KUKA KRL program: kuka_eki_command_serverB.sub, kuka_eki_command_serverB.dat

--- kuka_eki_command_serverB.sub ---
&ACCESS RVO1
&PARAM EDITMASK = *
&PARAM TEMPLATE = C:\KRC\Roboter\Template\submit
def kuka_eki_command_serverB()
   ;FOLD DECLARATIONS
   ;FOLD USER DECL
   ; local vairable declarations
   decl int elements_read

   eki_hw_iface_init() ; socket connection

   parameters[1] = $POS_ACT.X
   parameters[2] = $POS_ACT.Y
   parameters[3] = $POS_ACT.Z
   parameters[4] = $POS_ACT.A
   parameters[5] = $POS_ACT.B
   parameters[6] = $POS_ACT.C

   loop
      instruction_code = 0 ; reset instruction code to default
      elements_read = eki_hw_iface_get()  ; Get new command from buffer

      SWITCH (instruction_code)
      CASE 1
         ; cartesian motion XYZ command, phrase parameters into global variable cartesian_target
         cartesian_target.X = parameters[1]
         cartesian_target.Y = parameters[2]
         cartesian_target.Z = parameters[3]
         MsgNotify("Cartesian target XYZ command received and set",,,,)

      CASE 2
         ; cartesian motion XYZABC command
         cartesian_target.X = parameters[1]
         cartesian_target.Y = parameters[2]
         cartesian_target.Z = parameters[3]
         cartesian_target.A = parameters[4]
         cartesian_target.B = parameters[5]
         cartesian_target.C = parameters[6]

      CASE 3
         ; whether motion complete (0/1)
         json_motion_complete = parameters[1]

      CASE 4
         ; set linear velocity
         $VEL.CP = parameters[1]

      CASE 5
         ; set swivel velocity
         $VEL.ORI1 = parameters[1]

      CASE 6
         ; set swivel velocity
         $VEL.ORI2 = parameters[1]

      CASE 7
         LaserOff()
      CASE 8
         LaserOn()
      CASE 9
         LaserEnd()
      CASE 10
         LaserStart()
      CASE 11
         $ANOUT[1] = parameters[1] ; set laser power
      CASE 12
         $TOOL=TOOL_DATA[parameters[1]] ; set tool
      CASE 13
         $BASE.X = parameters[1]
         $BASE.Y = parameters[2]
         $BASE.Z = parameters[3]
         $BASE.A = parameters[4]
         $BASE.B = parameters[5]
         $BASE.C = parameters[6]
      CASE 14
         ;wait time between move
         wait_time = parameters[1]


      DEFAULT
         cartesian_target.X = $POS_ACT.X
         cartesian_target.Y = $POS_ACT.Y
         cartesian_target.Z = $POS_ACT.Z
         cartesian_target.A = $POS_ACT.A
         cartesian_target.B = $POS_ACT.B
         cartesian_target.C = $POS_ACT.C
      ENDSWITCH
   endloop


end



def eki_hw_iface_init()
   decl eki_status eki_ret

   ; Setup interrupts
   ; Interrupt 15 - Connection cleanup on client disconnect
   global interrupt decl 15 when $flag[1]==false do eki_hw_iface_reset()
   interrupt on 15
   ; Interrupt 16 - Timer interrupt for periodic state transmission
   global interrupt decl 16 when $timer_flag[1]==true do eki_hw_iface_send()
   interrupt on 16
   wait sec 0.012          ; Wait for next interpolation cycle
   $timer[1] = -200        ; Time in [ms] before first interrupt call
   $timer_stop[1] = false  ; Start timer 1

   ; Create and open EKI interface
   eki_ret = eki_init("EkiCommandServerB")
   eki_ret = eki_open("EkiCommandServerB")
   MsgNotify("ROS connection established",,,,)
end



def eki_hw_iface_send()
   decl eki_status eki_ret

   if $flag[1] then  ; If connection alive
      ; Load state values into xml structure
      ; position
      eki_ret = eki_setreal("EkiCommandServerB", "RobotState/Pos/@A1", $axis_act_meas.a1)
      eki_ret = eki_setreal("EkiCommandServerB", "RobotState/Pos/@A2", $axis_act_meas.a2)
      eki_ret = eki_setreal("EkiCommandServerB", "RobotState/Pos/@A3", $axis_act_meas.a3)
      eki_ret = eki_setreal("EkiCommandServerB", "RobotState/Pos/@A4", $axis_act_meas.a4)
      eki_ret = eki_setreal("EkiCommandServerB", "RobotState/Pos/@A5", $axis_act_meas.a5)
      eki_ret = eki_setreal("EkiCommandServerB", "RobotState/Pos/@A6", $axis_act_meas.a6)

      eki_ret = eki_setreal("EkiCommandServerB", "RobotState/Eff/@A1", $torque_axis_act[1])
      eki_ret = eki_setreal("EkiCommandServerB", "RobotState/Eff/@A2", $torque_axis_act[2])
      eki_ret = eki_setreal("EkiCommandServerB", "RobotState/Eff/@A3", $torque_axis_act[3])
      eki_ret = eki_setreal("EkiCommandServerB", "RobotState/Eff/@A4", $torque_axis_act[4])
      eki_ret = eki_setreal("EkiCommandServerB", "RobotState/Eff/@A5", $torque_axis_act[5])
      eki_ret = eki_setreal("EkiCommandServerB", "RobotState/Eff/@A6", $torque_axis_act[6])
      ; interface state
      eki_ret = eki_checkbuffer("EkiCommandServerB", "CommandServer/@InstructionCode")
      eki_ret = eki_setint("EkiCommandServerB", "RobotState/CommandServer/@Size", eki_ret.buff)

      ; Send xml structure
      if $flag[1] then  ; Make sure connection hasn't died while updating xml structure
         eki_ret = eki_send("EkiCommandServerB", "RobotState")
      endif
   endif

   ; Set timer for next interrupt [ms]
   $timer[1] = -10  ; ~10 ms for above send + 10 ms interrupt timer -> ~50 Hz state transmission
end


; eki_hw_iface_get: phrase command
; Tries to read most recent message from buffer. q left unchanged if empty.
; Returns number of elements read.
deffct int eki_hw_iface_get()
   decl eki_status eki_ret

   if not $flag[1] then
      return 0
   endif

   eki_ret = eki_checkbuffer("EkiCommandServerB", "CommandServer/@InstructionCode")
   if eki_ret.buff <= 0 then
     return 0
   endif

   eki_ret = eki_getint("EkiCommandServerB", "CommandServer/@InstructionCode", instruction_code)
   eki_ret = eki_getreal("EkiCommandServerB", "CommandServer/Parameters/@P1", parameters[1])
   eki_ret = eki_getreal("EkiCommandServerB", "CommandServer/Parameters/@P2", parameters[2])
   eki_ret = eki_getreal("EkiCommandServerB", "CommandServer/Parameters/@P3", parameters[3])
   eki_ret = eki_getreal("EkiCommandServerB", "CommandServer/Parameters/@P4", parameters[4])
   eki_ret = eki_getreal("EkiCommandServerB", "CommandServer/Parameters/@P5", parameters[5])
   eki_ret = eki_getreal("EkiCommandServerB", "CommandServer/Parameters/@P6", parameters[6])

   return 1
endfct


def eki_hw_iface_reset()
   decl eki_status eki_ret

   eki_ret = eki_clear("EkiCommandServerB")
   eki_ret = eki_init("EkiCommandServerB")
   eki_ret = eki_open("EkiCommandServerB")
end

--- kuka_eki_command_serverB.dat ---
&ACCESS RVO1
&PARAM EDITMASK = *
&PARAM TEMPLATE = C:\KRC\Roboter\Template\submit
defdat kuka_eki_command_serverB public
;FOLD EXTERNAL DECLARATIONS;%{PE}%MKUKATPBASIS,%CEXT,%VCOMMON,%P
;FOLD BASISTECH EXT;%{PE}%MKUKATPBASIS,%CEXT,%VEXT,%P
EXT  BAS (BAS_COMMAND  :IN,REAL  :IN )
DECL INT SUCCESS
;ENDFOLD (BASISTECH EXT)
;FOLD USER EXT;%{E}%MKUKATPUSER,%CEXT,%VEXT,%P
;Make your modifications here

;ENDFOLD (USER EXT)
;ENDFOLD (EXTERNAL DECLARATIONS)
decl global INT instruction_code = 0          ; identify which command (i.e, velocity, motion, laser, etc)
decl global real parameters[6]                ; number of received parameters in real value
decl global real json_motion_complete = 0     ; json motion command complete or not
decl global real wait_time = 0                ; wait time between move
parameters[1] = 0
decl global frame cartesian_target            ; frame is a sturct, X, Y, Z, A, B, C
;decl global pos cartesian_target_pos          ;pos: X, Y, Z, A, B, C, INT S, T
enddat
